{attribute 'GeneratedUsingTerminal: EL3783-0000-0018'}
{attribute addProperty BoxType "EL3783-0000-0018"}
{attribute addProperty Id "High_Current_RangeAT %I*High_Current_Range_489677624High_Current_Range_ActiveAT %I*BOOL1"}
{attribute addProperty CRC "2649480813"}
{attribute addProperty Size "5"}
TYPE AI_Current_Range_9DEBDE6D :
STRUCT
	{attribute addProperty Name "High_Current_Range"}
	High_Current_Range AT %I* : High_Current_Range_48967762;
	{attribute addProperty Name "High_Current_Range_Active"}
	High_Current_Range_Active AT %I* : BOOL;
END_STRUCT
END_TYPE

(* stored: Version 1.2.0.0, ProductVersion 3.1.4024.9
   DUT AI_Current_Range_9DEBDE6D: Id {4f628365-ceac-4464-b189-ff161b87d3ec} *)
